(* PLC project STAS-60.project, Eaton Automation XSOFT-CODESYS-3 - PLC programming system (Demo license) XSOFT-CODESYS V3.5.11 *)
(* stored: creationDateTime 2018-06-18T11:39:30.2804468, modificationDateTime 2018-06-18T10:33:33.3344536 *)

{attribute 'qualified_only'}
VAR_GLOBAL  (* GVL *)
  hiPres AT %IW2 : WORD;
  lowPres AT %IW4 : WORD;
  mowAbsorb AT %IW6 : WORD;
  lowPresAbsorb AT %IW8 : WORD;
  hiPresAbsorb AT %IW10 : WORD;
  nProcess : INT;
  kokoetoChislo : WORD;
END_VAR
